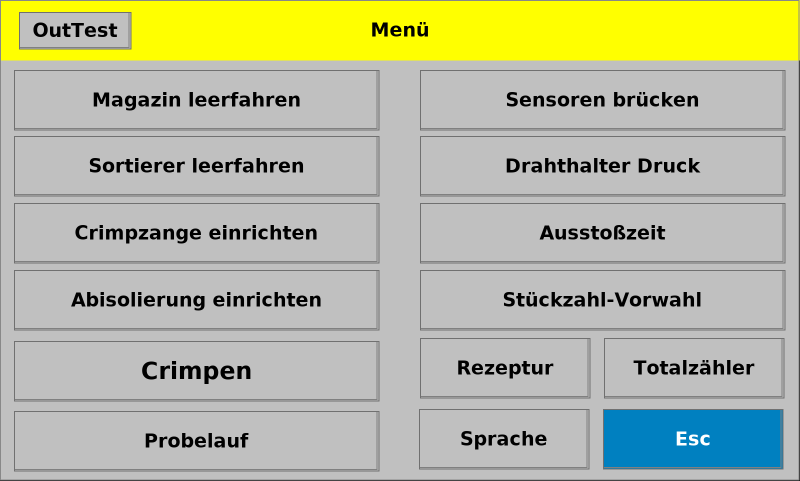
VISUALIZATION Menu  // 800x481
    Rectangle (0,1 800x480)
    Rectangle (0,0 800x60), "Menü"
        OnMouseUp: change screen: IO_Visu01
    Button (14,70 365x60), "Magazin leerfahren"
        OnMouseClick: execute { F_AuswertungBefehlstastenVonTP(tastenWert := CVL.MAGAZIN_LEER); }
        OnMouseUp: change screen: Start
    Button (14,136 365x60), "Sortierer leerfahren"
        OnMouseClick: execute { F_AuswertungBefehlstastenVonTP(tastenWert := CVL.SORTIER_LEER); }
        OnMouseUp: change screen: Start
    Button (14,203 365x60), "Crimpzange einrichten"
        OnMouseClick: execute { F_AuswertungBefehlstastenVonTP(tastenWert := CVL.CRIMP_EINRICHTEN); }
        OnMouseUp: change screen: Start
    Button (14,270 365x60), "Abisolierung einrichten"
        OnMouseClick: execute { F_AuswertungBefehlstastenVonTP(tastenWert := CVL.NUR_ABISOLIER); }
        OnMouseUp: change screen: Start
    Button (14,341 365x60), "Crimpen"
        OnMouseClick: execute { F_AuswertungBefehlstastenVonTP(tastenWert := CVL.RESET_BUTTON); F_ResetEndSchalterFehler(); }
        OnMouseUp: change screen: Start
    Button (14,411 365x60), "Probelauf"
        OnMouseUp: change screen: Probelauf
    Button (420,70 365x60), "Sensoren brücken"
        OnMouseClick: execute { GVL.EinzelschrittIdx := 500; }
        OnMouseUp: change screen: SensorBruecken
    Button (420,136 365x60), "Drahthalter Druck"
        OnMouseUp: change screen: DrahthalterDruck
    Button (420,203 365x60), "Ausstoßzeit"
        OnMouseUp: change screen: Ausstossverz
    Button (420,270 365x60), "Stückzahl-Vorwahl"
        OnMouseUp: change screen: Stueckzahl
    Button (420,338 170x60), "Rezeptur"
    Button (604,338 180x60), "Totalzähler"
        OnMouseUp: change screen: Total
    Button (419,409 170x60), "Sprache"
        OnMouseUp: change screen: Sprache
    Button (603,409 180x60), "Esc"
        OnMouseUp: change screen: Start
    Button (19,12 112x37), "OutTest"
        OnMouseUp: change screen: OutTest
END_VISUALIZATION

(* stored: Version 1.1.0.1, ProductVersion 3.1.4024.3
   Visu Menu: Id {b58000a8-7d35-4dbd-aa3d-173b78d7a2c2} *)
